FUNCTION_BLOCK FB_ClampSimulated
VAR_INPUT
	
END_VAR
VAR_OUTPUT
END_VAR
VAR
m_csState : CLAMP_STATE;	
m_csStateRequested : CLAMP_STATE;

//Eingänge
m_bIsOpen : BOOL;
m_bIsClosed : BOOL;
m_bIsClosedFull : BOOL;

//Ausgänge
m_bOpen :BOOL;
m_bClose :BOOL;

iWaitingTime : INT := 500;
iTimer: INT := 0;

END_VAR


StateMachine();

METHOD IsClosed : BOOL
VAR_INPUT
END_VAR

VAR
END_VAR
iTimer := iTimer +1;

IF iTimer > iWaitingTime THEN
	m_bIsClosed := TRUE;
	iTimer := 0;	
END_IF

IF m_csState = CLAMP_STATE.e_CLOSED THEN
	IsClosed := TRUE;
END_IF
END_METHOD

METHOD IsClosedFull : BOOL
VAR_INPUT
END_VAR

VAR
END_VAR

iTimer := iTimer +1;

IF iTimer > iWaitingTime THEN
	m_bIsClosedFull := TRUE;
	iTimer := 0;	
END_IF

IF m_csState = CLAMP_STATE.e_CLOSED_FULL THEN
	IsClosedFull := TRUE;
END_IF
END_METHOD

METHOD IsError : BOOL
VAR_INPUT
END_VAR
IF m_csState = CLAMP_STATE.e_ERROR THEN
	IsError := TRUE;
END_IF
END_METHOD

METHOD IsOpen : BOOL
VAR_INPUT
END_VAR

VAR
END_VAR
iTimer := iTimer +1;

IF iTimer > iWaitingTime THEN
	m_bIsOpen := TRUE;
	iTimer := 0;	
END_IF

IF m_csState = CLAMP_STATE.e_OPEN THEN
	IsOpen := TRUE;
END_IF
END_METHOD

METHOD SetCloseClampEmpty : BOOL
VAR_INPUT
END_VAR
m_csStateRequested := CLAMP_STATE.e_CLOSED;
m_bClose := TRUE;
SetCloseClampEmpty:=TRUE;
END_METHOD

METHOD SetCloseClampFull : BOOL
VAR_INPUT
END_VAR
m_csStateRequested := CLAMP_STATE.e_CLOSED_FULL;
m_bClose := TRUE;
SetCloseClampFull := TRUE;
END_METHOD

METHOD SetOpenClamp : BOOL
VAR_INPUT
END_VAR
m_bOpen := TRUE;
END_METHOD

METHOD StateMachine : BOOL
VAR_INPUT
END_VAR

//m_bIsOpen : BOOL;
//m_bIsClosed : BOOL;
//m_bIsClosedFull : BOOL;

CASE m_csState  OF
	
	CLAMP_STATE.e_OPEN:	
		

		IF m_bIsClosed THEN
			m_csState := CLAMP_STATE.e_CLOSED;		
		END_IF
		
		IF m_bIsClosedFull THEN
			m_csState := CLAMP_STATE.e_CLOSED_FULL;		
		END_IF
		
 	CLAMP_STATE.e_CLOSED_FULL:
	// Fehler wenn falscher Zustand
 		IF m_csStateRequested = CLAMP_STATE.e_CLOSED THEN
  			m_csState := CLAMP_STATE.e_ERROR;
		END_IF
		
		
		IF m_bIsOpen THEN
			m_csState := CLAMP_STATE.e_OPEN;		
		END_IF
	
	CLAMP_STATE.e_CLOSED:
			// Fehler wenn falscher Zustand in diesem Fall: Werkstück erwartet aber nicht im Halter
 		IF m_csStateRequested = CLAMP_STATE.e_CLOSED_FULL THEN
  			m_csState := CLAMP_STATE.e_ERROR;
		END_IF
	
	
		IF m_bIsOpen THEN
			m_csState := CLAMP_STATE.e_OPEN;		
		END_IF
		
CLAMP_STATE.e_ERROR:
		
END_CASE
END_METHOD

END_FUNCTION_BLOCK

(* stored: Version 1.1.0.1, ProductVersion 3.1.4024.0
   POU FB_ClampSimulated: Id {c069c4d4-a266-429b-b0eb-1149e80b5f6d}, SpecialFunc None
   Method IsClosed: Id {118c5ee9-937f-4215-9d0e-097c74a007e1}
   Method IsClosedFull: Id {f65ce7cb-9130-48d2-bf35-af4fc1162e6a}
   Method IsError: Id {51d77b77-8199-4dc2-813b-d8c4997239e3}
   Method IsOpen: Id {49c32a2f-6a54-4b35-9a2a-5c49ca470baf}
   Method SetCloseClampEmpty: Id {bfdd8289-4452-4488-b6ed-2ebfdaef12b1}
   Method SetCloseClampFull: Id {082f351c-b7ea-4125-b5c5-15893bc06490}
   Method SetOpenClamp: Id {37be77fd-6a2e-46f4-8fd3-00e4562e41a5}
   Method StateMachine: Id {84584eb1-8243-4da9-9d15-4bf3edc14468} *)
